// TIA Portal V17 export
// export: Created 2022-07-20T06:59:50.6311915Z, ExportSetting WithDefaults, DisplayName Totally Integrated Automation Portal, DisplayVersion V17, DisplayName TIA Portal Openness, DisplayVersion V17, DisplayName TIA Portal Version Control Interface, DisplayVersion V17, DisplayName SINAMICS Startdrive Advanced, DisplayVersion V17, DisplayName SINAMICS Startdrive G130, G150, S120, S150, SINAMICS MV, S210, DisplayVersion V17, DisplayName SINAMICS Startdrive G110M, G120, G120C, G120D, G120P, G115D, DisplayVersion V17, DisplayName STEP 7 Professional, DisplayVersion V17, DisplayName STEP 7 Safety, DisplayVersion V17, DisplayName WinCC Advanced, DisplayVersion V17
FUNCTION_BLOCK "FB10061_IperAirCircuit"   // FB10061, LAD
{ S7_Optimized_Access := 'TRUE' }
VERSION : 0.1
// stored: AutoNumber false, IsIECCheckEnabled false, IsRetainMemResEnabled false, MemoryReserve 100, SetENOAutomatically false, UDAEnableTagReadback false
   VAR_INPUT
      ManometerSetPoint : Real;
      ManometerRawValue : Real;
   END_VAR
   VAR_OUTPUT
      InError : Bool;
      PressurizatonDone : Bool;
      DepressurizatonDone : Bool;
      ManometerPressurePower : Int;
      ManometerActualPressure : Real;
   END_VAR
   VAR_IN_OUT
      RequestAcknowledge : Bool;
      RequestPressurization : Bool;
      RequestDepressurization : Bool;
   END_VAR
   VAR
      IperAirOperationStateDiagram : Int;
      R_TRIG_RequestPressurization : R_TRIG;
      R_TRIG_RequestDepressurization { S7_SetPoint := 'True'} : R_TRIG;
      F_TRIG_RequestPressurization { S7_SetPoint := 'True'} : F_TRIG;
      F_TRIG_RequestDepressurization { S7_SetPoint := 'True'} : F_TRIG;
      TON_PressurizationTiming { S7_SetPoint := 'True'} : TON_TIME;
   END_VAR
   VAR CONSTANT
      WAIT_FOR_FOR_OPERATION_REQUEST : Int := 0;
      PRESSURIZATION : Int := 10;
      DEPRESSURIZATION : Int := 20;
      OPERATION_DONE : Int := 30;
   END_VAR
BEGIN

REGION Network 1 (SCL): First Scan
   IF
       "FirstScan"
   THEN
       #IperAirOperationStateDiagram := #WAIT_FOR_FOR_OPERATION_REQUEST;
       #PressurizatonDone := FALSE;
       #DepressurizatonDone := FALSE;
   END_IF;
END_REGION

REGION Network 2 (SCL): Edge Signals & Timer
   REGION EDGE SIGNALS
       #R_TRIG_RequestPressurization(CLK := #RequestPressurization);
       #R_TRIG_RequestDepressurization(CLK := #RequestDepressurization);

       #F_TRIG_RequestPressurization(CLK := #RequestPressurization);
       #F_TRIG_RequestDepressurization(CLK := #RequestDepressurization);
   END_REGION

   REGION TIMER
       #TON_PressurizationTiming(IN := #IperAirOperationStateDiagram = #PRESSURIZATION,
                                 PT := T#10s);
   END_REGION
END_REGION

REGION Network 3 (SCL): Pressurization management
   CASE #IperAirOperationStateDiagram OF
       #WAIT_FOR_FOR_OPERATION_REQUEST:
           IF #R_TRIG_RequestPressurization.Q THEN
               #PressurizatonDone := FALSE;
               #DepressurizatonDone := FALSE;
               #IperAirOperationStateDiagram := #PRESSURIZATION;
           ELSIF #R_TRIG_RequestDepressurization.Q THEN
               #PressurizatonDone := FALSE;
               #DepressurizatonDone := FALSE;
               #IperAirOperationStateDiagram := #DEPRESSURIZATION;
           END_IF;
       #PRESSURIZATION:
           #ManometerPressurePower := REAL_TO_INT(#ManometerSetPoint);
           IF "FC10021_TolerenceRelation"(X := #ManometerRawValue, Y := #ManometerSetPoint, Tolerance := 5.0) THEN
               #RequestPressurization := FALSE;
               #PressurizatonDone := TRUE;
               #IperAirOperationStateDiagram := #OPERATION_DONE;
           ELSIF #TON_PressurizationTiming.Q THEN
               #IperAirOperationStateDiagram := #OPERATION_DONE;
           END_IF;
       #DEPRESSURIZATION:
           #ManometerPressurePower := 0;
           IF #ManometerRawValue = 0.0 THEN
               #RequestDepressurization := FALSE;
               #DepressurizatonDone := TRUE;
               #IperAirOperationStateDiagram := #OPERATION_DONE;
           END_IF;
       #OPERATION_DONE:
           #IperAirOperationStateDiagram := #WAIT_FOR_FOR_OPERATION_REQUEST;
   END_CASE;
END_REGION

REGION Network 4 (SCL): Iper Air Circuit States Management
   #ManometerActualPressure := #ManometerRawValue;
END_REGION

REGION Network 5 (SCL): Error Management
   IF #TON_PressurizationTiming.Q THEN
       #InError := TRUE;
   ELSIF #RequestAcknowledge THEN
       #InError := FALSE;
   END_IF;
END_REGION
END_FUNCTION_BLOCK
